# EPICS autosave request: URModuleApp/Db/set_movement_params_settings.req
$(P)$(R)MoveParams:TCPOffset_X.VAL
$(P)$(R)MoveParams:TCPOffset_Y.VAL
$(P)$(R)MoveParams:TCPOffset_Z.VAL
$(P)$(R)MoveParams:TCPOffset_Roll.VAL
$(P)$(R)MoveParams:TCPOffset_Pitch.VAL
$(P)$(R)MoveParams:TCPOffset_Yaw.VAL
$(P)$(R)MoveParams:Velocity.VAL
$(P)$(R)MoveParams:GripperSpeed.VAL
$(P)$(R)MoveParams:GripperForce.VAL
